// TIA Portal V18 export
TYPE "LGasp_StatoAttuatori"
// stored: IsFailsafeCompliant false
   STRUCT
      attuatore { ExternalWritable := 'False'} : Array[1.."N_MaxAttuatoriStz"] of "LGasp_typeStatoAttuatore";
   END_STRUCT;
END_TYPE
